{attribute 'qualified_only'}
{attribute 'strict'}
{attribute 'to_string'}
TYPE E_HomeStates :
(
    IDLE:= 0,
    NEXT_MOVE:= 1,
    CHECK_FWD:= 2,
    CHECK_BWD:= 3,
    FINAL_MOVE:= 4,
    FINAL_SETPOS:= 5,
    ERROR:= -99,
    WAIT_STOP:= 7
) INT;
END_TYPE

(* stored: Version 1.1.0.1
   DUT E_HomeStates: Id {1da1e1be-06ef-4806-abac-49565ed1ebca} *)
